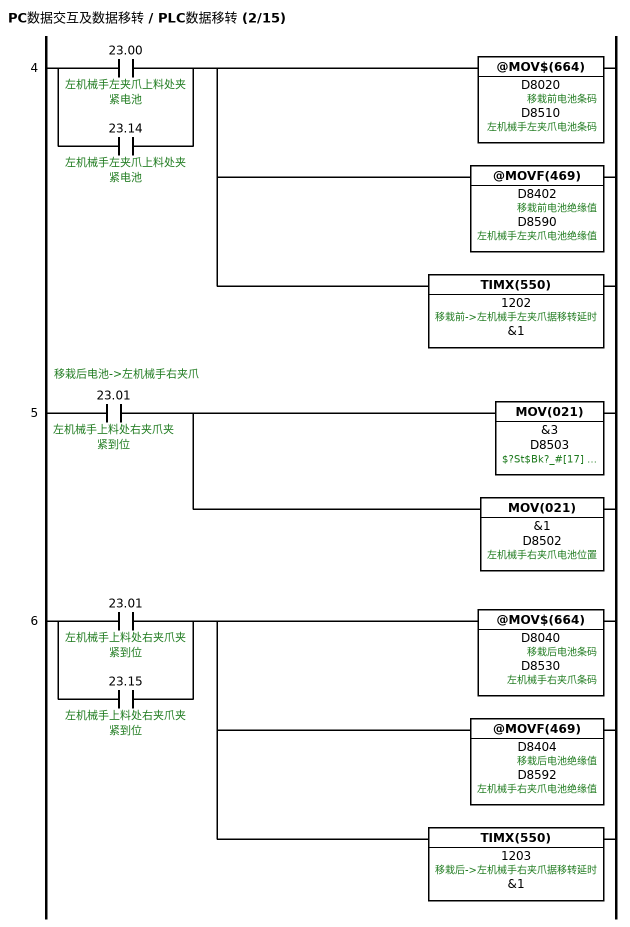
; [picture p425: PC数据交互及数据移转 / PLC数据移转, rungs 4-6]
; rung 4
LD 23.00  ; 左机械手左夹爪上料处夹紧电池
OR 23.14  ; 左机械手左夹爪上料处夹紧电池
@MOV$(664) D8020 D8510  ; 移栽前电池条码, 左机械手左夹爪电池条码
@MOVF(469) D8402 D8590  ; 移栽前电池绝缘值, 左机械手左夹爪电池绝缘值
TIMX(550) 1202 &1  ; 移栽前->左机械手左夹爪据移转延时
; rung 5: 移栽后电池->左机械手右夹爪
LD 23.01  ; 左机械手上料处右夹爪夹紧到位
MOV(021) &3 D8503  ; $?St$Bk?_#[17] / 左机械手右夹爪电池结果$?St$Bk?_#[17]
MOV(021) &1 D8502  ; 左机械手右夹爪电池位置
; rung 6
LD 23.01  ; 左机械手上料处右夹爪夹紧到位
OR 23.15  ; 左机械手上料处右夹爪夹紧到位
@MOV$(664) D8040 D8530  ; 移栽后电池条码, 左机械手右夹爪条码
@MOVF(469) D8404 D8592  ; 移栽后电池绝缘值, 左机械手右夹爪电池绝缘值
TIMX(550) 1203 &1  ; 移栽后->左机械手右夹爪据移转延时

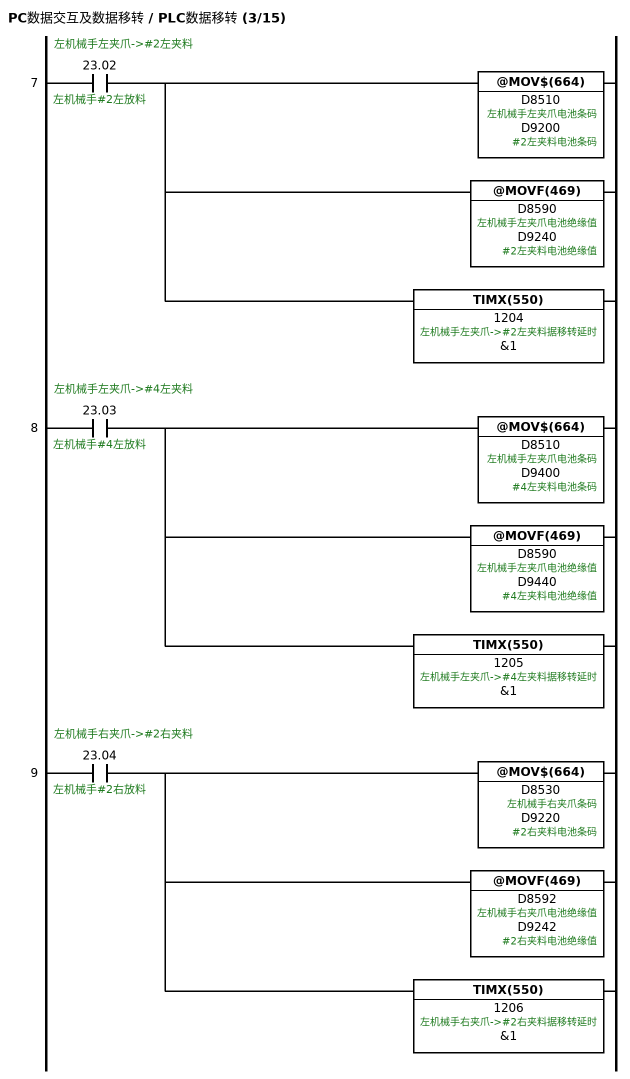
; rung 7: 左机械手左夹爪->#2左夹料
LD 23.02  ; 左机械手#2左放料
@MOV$(664) D8510 D9200  ; 左机械手左夹爪电池条码, #2左夹料电池条码
@MOVF(469) D8590 D9240  ; 左机械手左夹爪电池绝缘值, #2左夹料电池绝缘值
TIMX(550) 1204 &1  ; 左机械手左夹爪->#2左夹料据移转延时
; rung 8: 左机械手左夹爪->#4左夹料
LD 23.03  ; 左机械手#4左放料
@MOV$(664) D8510 D9400  ; 左机械手左夹爪电池条码, #4左夹料电池条码
@MOVF(469) D8590 D9440  ; 左机械手左夹爪电池绝缘值, #4左夹料电池绝缘值
TIMX(550) 1205 &1  ; 左机械手左夹爪->#4左夹料据移转延时
; rung 9: 左机械手右夹爪->#2右夹料
LD 23.04  ; 左机械手#2右放料
@MOV$(664) D8530 D9220  ; 左机械手右夹爪条码, #2右夹料电池条码
@MOVF(469) D8592 D9242  ; 左机械手右夹爪电池绝缘值, #2右夹料电池绝缘值
TIMX(550) 1206 &1  ; 左机械手右夹爪->#2右夹料据移转延时

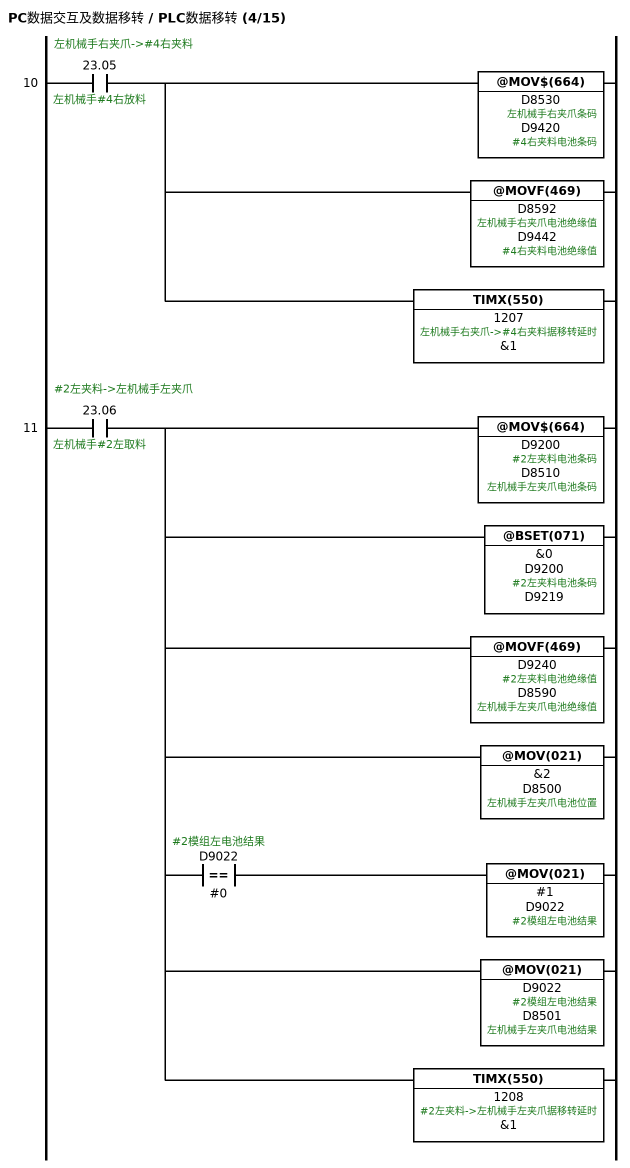
; rung 10: 左机械手右夹爪->#4右夹料
LD 23.05  ; 左机械手#4右放料
@MOV$(664) D8530 D9420  ; 左机械手右夹爪条码, #4右夹料电池条码
@MOVF(469) D8592 D9442  ; 左机械手右夹爪电池绝缘值, #4右夹料电池绝缘值
TIMX(550) 1207 &1  ; 左机械手右夹爪->#4右夹料据移转延时
; rung 11: #2左夹料->左机械手左夹爪
LD 23.06  ; 左机械手#2左取料
OUT TR0
@MOV$(664) D9200 D8510  ; #2左夹料电池条码, 左机械手左夹爪电池条码
@BSET(071) &0 D9200 D9219  ; #2左夹料电池条码
@MOVF(469) D9240 D8590  ; #2左夹料电池绝缘值, 左机械手左夹爪电池绝缘值
@MOV(021) &2 D8500  ; 左机械手左夹爪电池位置
AND=(300) D9022 #0  ; #2模组左电池结果
@MOV(021) #1 D9022  ; #2模组左电池结果
LD TR0
@MOV(021) D9022 D8501  ; #2模组左电池结果, 左机械手左夹爪电池结果
TIMX(550) 1208 &1  ; #2左夹料->左机械手左夹爪据移转延时

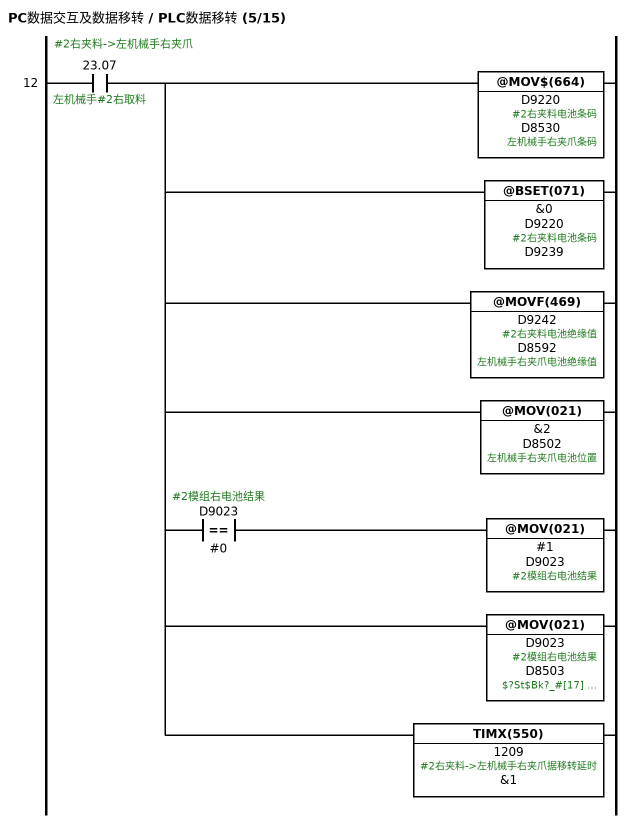
; rung 12: #2右夹料->左机械手右夹爪
LD 23.07  ; 左机械手#2右取料
OUT TR0
@MOV$(664) D9220 D8530  ; #2右夹料电池条码, 左机械手右夹爪条码
@BSET(071) &0 D9220 D9239  ; #2右夹料电池条码
@MOVF(469) D9242 D8592  ; #2右夹料电池绝缘值, 左机械手右夹爪电池绝缘值
@MOV(021) &2 D8502  ; 左机械手右夹爪电池位置
AND=(300) D9023 #0  ; #2模组右电池结果
@MOV(021) #1 D9023  ; #2模组右电池结果
LD TR0
@MOV(021) D9023 D8503  ; #2模组右电池结果, $?St$Bk?_#[17] / 左机械手右夹爪电池结果$?St$Bk?_#[17]
TIMX(550) 1209 &1  ; #2右夹料->左机械手右夹爪据移转延时

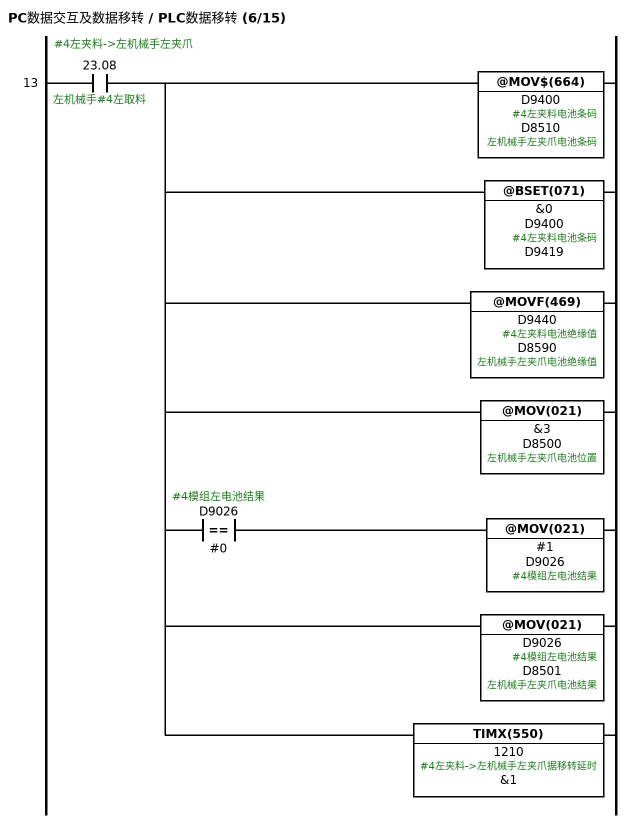
; rung 13: #4左夹料->左机械手左夹爪
LD 23.08  ; 左机械手#4左取料
OUT TR0
@MOV$(664) D9400 D8510  ; #4左夹料电池条码, 左机械手左夹爪电池条码
@BSET(071) &0 D9400 D9419  ; #4左夹料电池条码
@MOVF(469) D9440 D8590  ; #4左夹料电池绝缘值, 左机械手左夹爪电池绝缘值
@MOV(021) &3 D8500  ; 左机械手左夹爪电池位置
AND=(300) D9026 #0  ; #4模组左电池结果
@MOV(021) #1 D9026  ; #4模组左电池结果
LD TR0
@MOV(021) D9026 D8501  ; #4模组左电池结果, 左机械手左夹爪电池结果
TIMX(550) 1210 &1  ; #4左夹料->左机械手左夹爪据移转延时

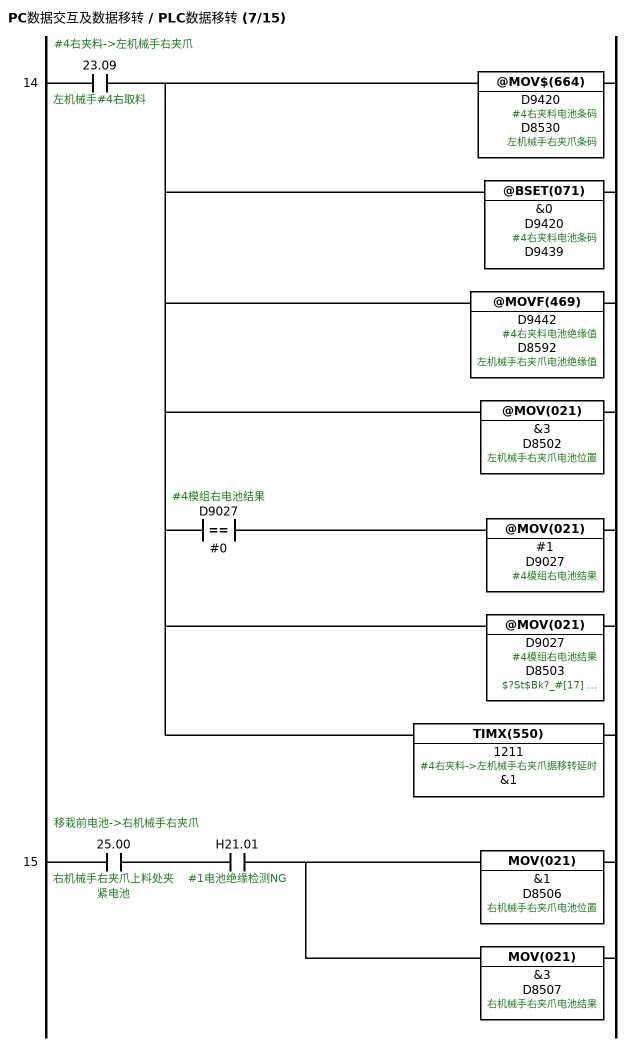
; rung 14: #4右夹料->左机械手右夹爪
LD 23.09  ; 左机械手#4右取料
OUT TR0
@MOV$(664) D9420 D8530  ; #4右夹料电池条码, 左机械手右夹爪条码
@BSET(071) &0 D9420 D9439  ; #4右夹料电池条码
@MOVF(469) D9442 D8592  ; #4右夹料电池绝缘值, 左机械手右夹爪电池绝缘值
@MOV(021) &3 D8502  ; 左机械手右夹爪电池位置
AND=(300) D9027 #0  ; #4模组右电池结果
@MOV(021) #1 D9027  ; #4模组右电池结果
LD TR0
@MOV(021) D9027 D8503  ; #4模组右电池结果, $?St$Bk?_#[17] / 左机械手右夹爪电池结果$?St$Bk?_#[17]
TIMX(550) 1211 &1  ; #4右夹料->左机械手右夹爪据移转延时
; rung 15: 移栽前电池->右机械手右夹爪
LD 25.00  ; 右机械手右夹爪上料处夹紧电池
AND H21.01  ; #1电池绝缘检测NG
MOV(021) &1 D8506  ; 右机械手右夹爪电池位置
MOV(021) &3 D8507  ; 右机械手右夹爪电池结果

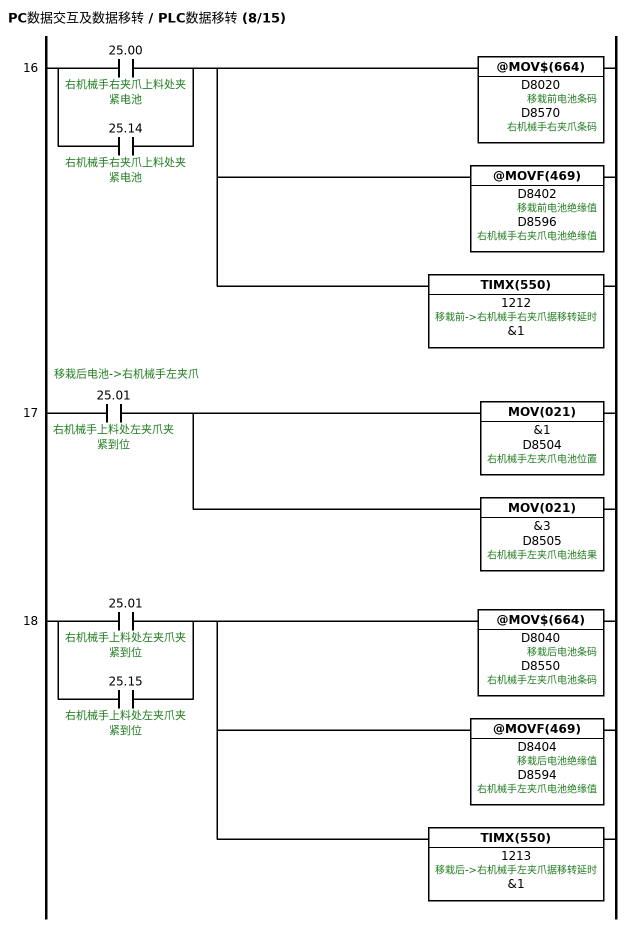
; rung 16
LD 25.00  ; 右机械手右夹爪上料处夹紧电池
OR 25.14  ; 右机械手右夹爪上料处夹紧电池
@MOV$(664) D8020 D8570  ; 移栽前电池条码, 右机械手右夹爪条码
@MOVF(469) D8402 D8596  ; 移栽前电池绝缘值, 右机械手右夹爪电池绝缘值
TIMX(550) 1212 &1  ; 移栽前->右机械手右夹爪据移转延时
; rung 17: 移栽后电池->右机械手左夹爪
LD 25.01  ; 右机械手上料处左夹爪夹紧到位
MOV(021) &1 D8504  ; 右机械手左夹爪电池位置
MOV(021) &3 D8505  ; 右机械手左夹爪电池结果
; rung 18
LD 25.01  ; 右机械手上料处左夹爪夹紧到位
OR 25.15  ; 右机械手上料处左夹爪夹紧到位
@MOV$(664) D8040 D8550  ; 移栽后电池条码, 右机械手左夹爪电池条码
@MOVF(469) D8404 D8594  ; 移栽后电池绝缘值, 右机械手左夹爪电池绝缘值
TIMX(550) 1213 &1  ; 移栽后->右机械手左夹爪据移转延时

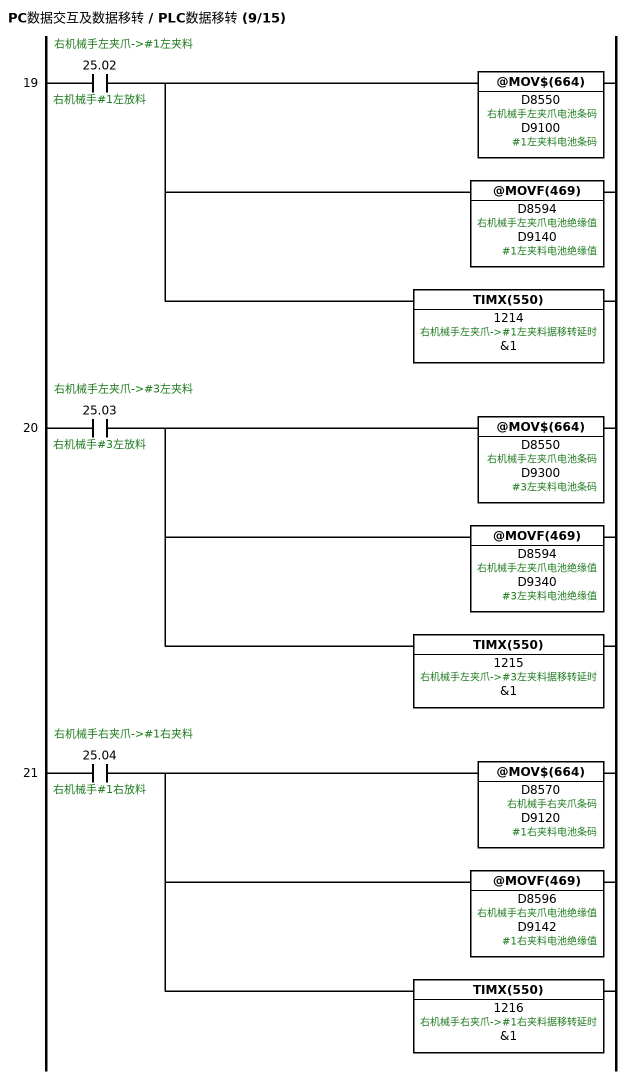
; rung 19: 右机械手左夹爪->#1左夹料
LD 25.02  ; 右机械手#1左放料
@MOV$(664) D8550 D9100  ; 右机械手左夹爪电池条码, #1左夹料电池条码
@MOVF(469) D8594 D9140  ; 右机械手左夹爪电池绝缘值, #1左夹料电池绝缘值
TIMX(550) 1214 &1  ; 右机械手左夹爪->#1左夹料据移转延时
; rung 20: 右机械手左夹爪->#3左夹料
LD 25.03  ; 右机械手#3左放料
@MOV$(664) D8550 D9300  ; 右机械手左夹爪电池条码, #3左夹料电池条码
@MOVF(469) D8594 D9340  ; 右机械手左夹爪电池绝缘值, #3左夹料电池绝缘值
TIMX(550) 1215 &1  ; 右机械手左夹爪->#3左夹料据移转延时
; rung 21: 右机械手右夹爪->#1右夹料
LD 25.04  ; 右机械手#1右放料
@MOV$(664) D8570 D9120  ; 右机械手右夹爪条码, #1右夹料电池条码
@MOVF(469) D8596 D9142  ; 右机械手右夹爪电池绝缘值, #1右夹料电池绝缘值
TIMX(550) 1216 &1  ; 右机械手右夹爪->#1右夹料据移转延时

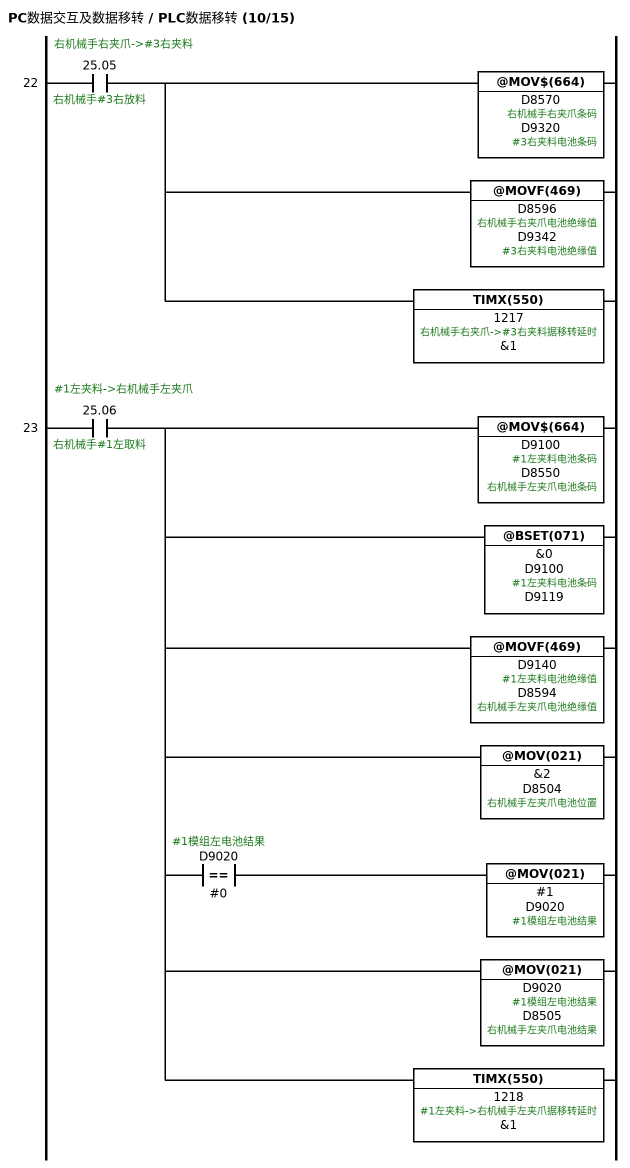
; rung 22: 右机械手右夹爪->#3右夹料
LD 25.05  ; 右机械手#3右放料
@MOV$(664) D8570 D9320  ; 右机械手右夹爪条码, #3右夹料电池条码
@MOVF(469) D8596 D9342  ; 右机械手右夹爪电池绝缘值, #3右夹料电池绝缘值
TIMX(550) 1217 &1  ; 右机械手右夹爪->#3右夹料据移转延时
; rung 23: #1左夹料->右机械手左夹爪
LD 25.06  ; 右机械手#1左取料
OUT TR0
@MOV$(664) D9100 D8550  ; #1左夹料电池条码, 右机械手左夹爪电池条码
@BSET(071) &0 D9100 D9119  ; #1左夹料电池条码
@MOVF(469) D9140 D8594  ; #1左夹料电池绝缘值, 右机械手左夹爪电池绝缘值
@MOV(021) &2 D8504  ; 右机械手左夹爪电池位置
AND=(300) D9020 #0  ; #1模组左电池结果
@MOV(021) #1 D9020  ; #1模组左电池结果
LD TR0
@MOV(021) D9020 D8505  ; #1模组左电池结果, 右机械手左夹爪电池结果
TIMX(550) 1218 &1  ; #1左夹料->右机械手左夹爪据移转延时

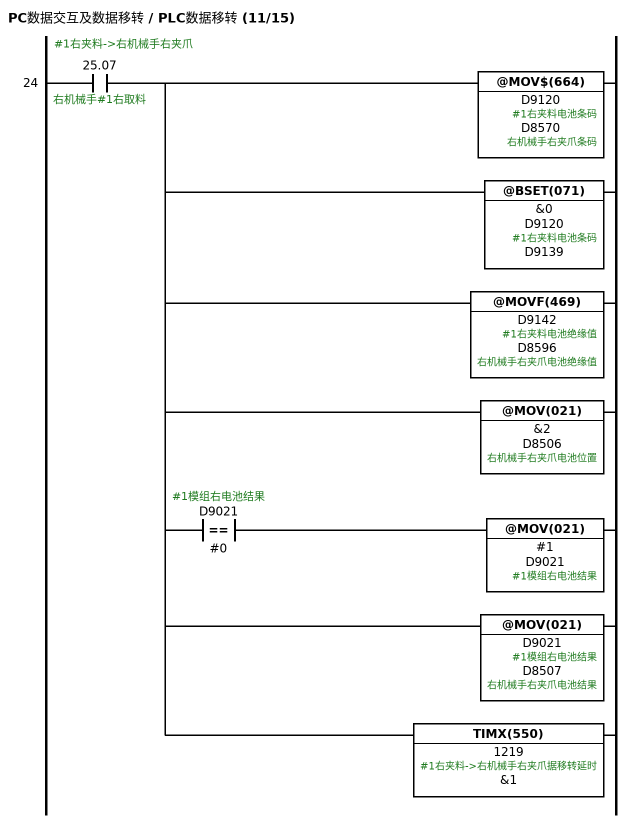
; rung 24: #1右夹料->右机械手右夹爪
LD 25.07  ; 右机械手#1右取料
OUT TR0
@MOV$(664) D9120 D8570  ; #1右夹料电池条码, 右机械手右夹爪条码
@BSET(071) &0 D9120 D9139  ; #1右夹料电池条码
@MOVF(469) D9142 D8596  ; #1右夹料电池绝缘值, 右机械手右夹爪电池绝缘值
@MOV(021) &2 D8506  ; 右机械手右夹爪电池位置
AND=(300) D9021 #0  ; #1模组右电池结果
@MOV(021) #1 D9021  ; #1模组右电池结果
LD TR0
@MOV(021) D9021 D8507  ; #1模组右电池结果, 右机械手右夹爪电池结果
TIMX(550) 1219 &1  ; #1右夹料->右机械手右夹爪据移转延时

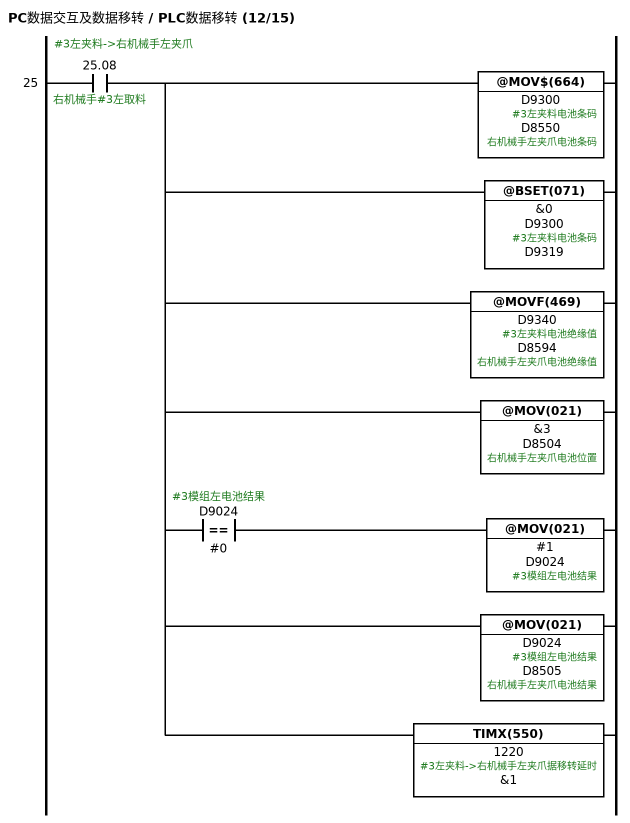
; rung 25: #3左夹料->右机械手左夹爪
LD 25.08  ; 右机械手#3左取料
OUT TR0
@MOV$(664) D9300 D8550  ; #3左夹料电池条码, 右机械手左夹爪电池条码
@BSET(071) &0 D9300 D9319  ; #3左夹料电池条码
@MOVF(469) D9340 D8594  ; #3左夹料电池绝缘值, 右机械手左夹爪电池绝缘值
@MOV(021) &3 D8504  ; 右机械手左夹爪电池位置
AND=(300) D9024 #0  ; #3模组左电池结果
@MOV(021) #1 D9024  ; #3模组左电池结果
LD TR0
@MOV(021) D9024 D8505  ; #3模组左电池结果, 右机械手左夹爪电池结果
TIMX(550) 1220 &1  ; #3左夹料->右机械手左夹爪据移转延时

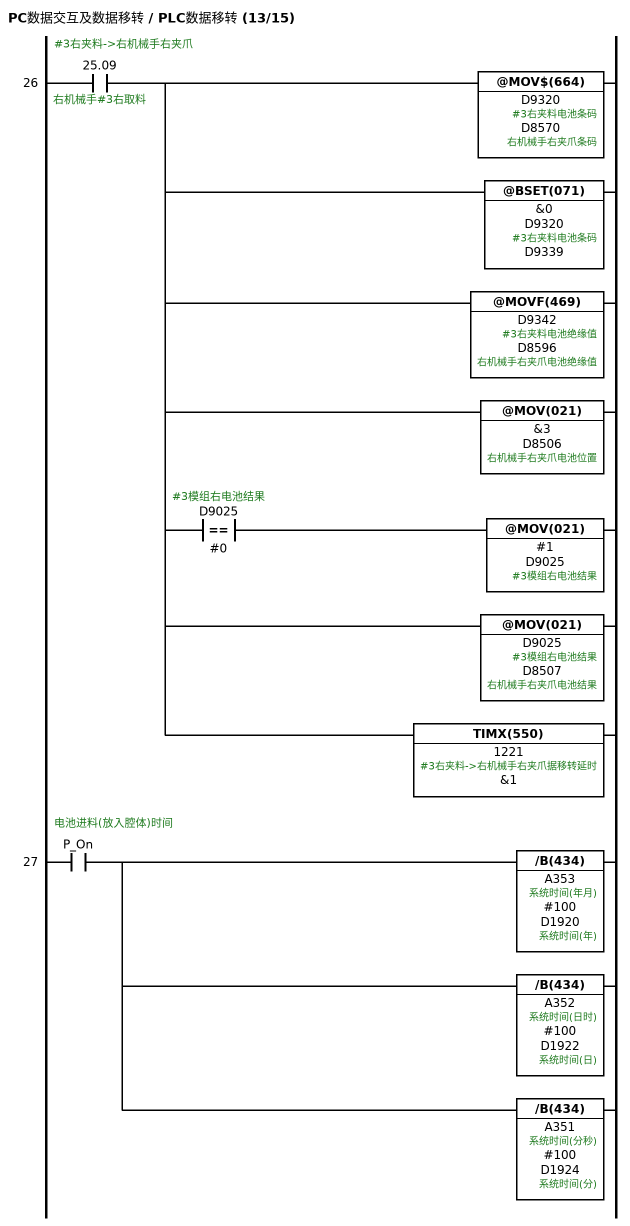
; rung 26: #3右夹料->右机械手右夹爪
LD 25.09  ; 右机械手#3右取料
OUT TR0
@MOV$(664) D9320 D8570  ; #3右夹料电池条码, 右机械手右夹爪条码
@BSET(071) &0 D9320 D9339  ; #3右夹料电池条码
@MOVF(469) D9342 D8596  ; #3右夹料电池绝缘值, 右机械手右夹爪电池绝缘值
@MOV(021) &3 D8506  ; 右机械手右夹爪电池位置
AND=(300) D9025 #0  ; #3模组右电池结果
@MOV(021) #1 D9025  ; #3模组右电池结果
LD TR0
@MOV(021) D9025 D8507  ; #3模组右电池结果, 右机械手右夹爪电池结果
TIMX(550) 1221 &1  ; #3右夹料->右机械手右夹爪据移转延时
; rung 27: 电池进料(放入腔体)时间
LD P_On
/B(434) A353 #100 D1920  ; 系统时间(年月), 系统时间(年)
/B(434) A352 #100 D1922  ; 系统时间(日时), 系统时间(日)
/B(434) A351 #100 D1924  ; 系统时间(分秒), 系统时间(分)

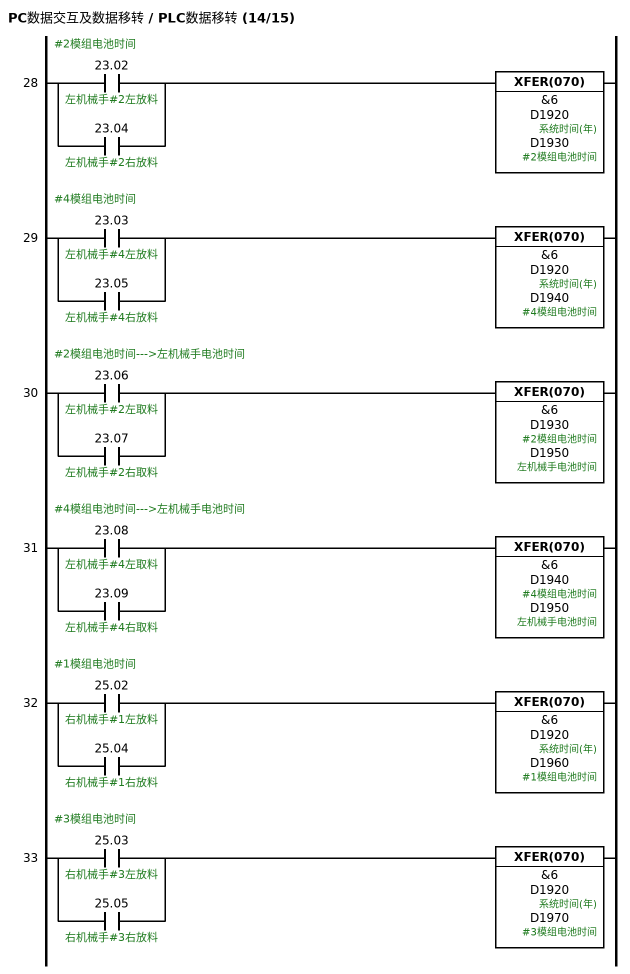
; rung 28: #2模组电池时间
LD 23.02  ; 左机械手#2左放料
OR 23.04  ; 左机械手#2右放料
XFER(070) &6 D1920 D1930  ; 系统时间(年), #2模组电池时间
; rung 29: #4模组电池时间
LD 23.03  ; 左机械手#4左放料
OR 23.05  ; 左机械手#4右放料
XFER(070) &6 D1920 D1940  ; 系统时间(年), #4模组电池时间
; rung 30: #2模组电池时间--->左机械手电池时间
LD 23.06  ; 左机械手#2左取料
OR 23.07  ; 左机械手#2右取料
XFER(070) &6 D1930 D1950  ; #2模组电池时间, 左机械手电池时间
; rung 31: #4模组电池时间--->左机械手电池时间
LD 23.08  ; 左机械手#4左取料
OR 23.09  ; 左机械手#4右取料
XFER(070) &6 D1940 D1950  ; #4模组电池时间, 左机械手电池时间
; rung 32: #1模组电池时间
LD 25.02  ; 右机械手#1左放料
OR 25.04  ; 右机械手#1右放料
XFER(070) &6 D1920 D1960  ; 系统时间(年), #1模组电池时间
; rung 33: #3模组电池时间
LD 25.03  ; 右机械手#3左放料
OR 25.05  ; 右机械手#3右放料
XFER(070) &6 D1920 D1970  ; 系统时间(年), #3模组电池时间

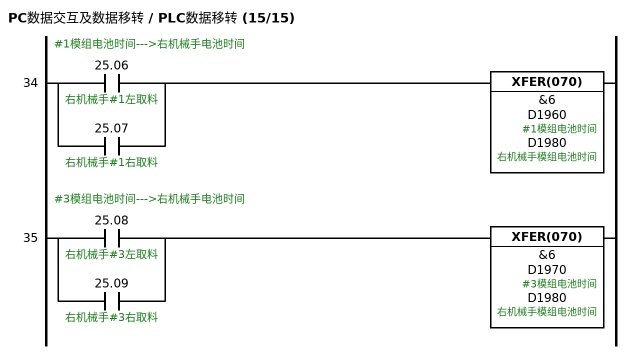
; rung 34: #1模组电池时间--->右机械手电池时间
LD 25.06  ; 右机械手#1左取料
OR 25.07  ; 右机械手#1右取料
XFER(070) &6 D1960 D1980  ; #1模组电池时间, 右机械手模组电池时间
; rung 35: #3模组电池时间--->右机械手电池时间
LD 25.08  ; 右机械手#3左取料
OR 25.09  ; 右机械手#3右取料
XFER(070) &6 D1970 D1980  ; #3模组电池时间, 右机械手模组电池时间

### Section END
; rung 0
END(001)